INTERFACE I_MotionAxisContinuous


METHOD MoveContinuous
VAR_INPUT
    Position	: LREAL;
    Velocity	: LREAL;
    Acceleration	: LREAL := 0.0;
    Deceleration	: LREAL := 0.0;
    Jerk	: LREAL := 0.0;
    BufferMode	: MC_BufferMode := .MC_BufferMode.MC_Aborting;
END_VAR
VAR_OUTPUT
    InVelocity	: BOOL;
    Busy	: BOOL;
    Active	: BOOL;
    CommandAborted	: BOOL;
    Error	: BOOL;
    ErrorID	: UDINT;
    ErrorStr	: T_MaxString;
END_VAR
END_METHOD

PROPERTY MoveContinuousBusy : BOOL
GET
END_GET
END_PROPERTY

PROPERTY MoveContinuousError : BOOL
GET
END_GET
END_PROPERTY

PROPERTY MoveContinuousErrorID : UDINT
GET
END_GET
END_PROPERTY

PROPERTY MoveContinuousInVelocity : BOOL
GET
END_GET
END_PROPERTY

PROPERTY MoveContinuousPassedTargetPosition : BOOL
GET
END_GET
END_PROPERTY

END_INTERFACE

(* stored: Version 1.1.0.1
   Itf I_MotionAxisContinuous: Id {9476e776-665e-453e-b113-3e0936768038}
   Method MoveContinuous: Id {b696eb2b-846c-4773-aec4-06e3ed4d56f2}
   Property MoveContinuousBusy: Id {99373bb0-4c47-434a-8ce1-627213de2e63}
   Get Get: Id {eee6f878-9445-40c6-b2b3-4295ace10728}
   Property MoveContinuousError: Id {ffedd637-58da-470b-bb0a-c4ae7c578290}
   Get Get: Id {2a141798-1efe-48d6-b310-6365edf3982c}
   Property MoveContinuousErrorID: Id {d785703c-8cf6-4e72-95fe-eec1a8deb29e}
   Get Get: Id {424c0687-5ecd-43f3-a318-678bad488a14}
   Property MoveContinuousInVelocity: Id {66092af1-db75-4204-a630-5d16e74e05fb}
   Get Get: Id {6191e831-8624-44f0-8de7-493ff650818d}
   Property MoveContinuousPassedTargetPosition: Id {9b2e0d90-11d1-4cb4-8740-ef840221c736}
   Get Get: Id {9a3b3169-b6df-4247-b68d-c70f792005c7} *)
